# EPICS substitutions: ek9000App/Db/EL1114.substitutions
file EL1114.template
{       pattern
        {
                TERMINAL,

        }
        {
        }
}
